PROPERTY PUBLIC p_PosR : REAL
GET
p_PosR := _Pos_R;
END_GET
END_PROPERTY

PROPERTY PUBLIC p_PosW : REAL
GET
p_PosW := _Pos_W;
END_GET
END_PROPERTY

PROPERTY PUBLIC p_PosX : REAL
GET
p_PosX := _Pos_X;
END_GET
END_PROPERTY

PROPERTY PUBLIC p_PosY : REAL
GET
p_PosY := _Pos_Y;
END_GET
END_PROPERTY

PROPERTY PUBLIC p_PosZ : REAL
GET
p_PosZ := _Pos_Z;
END_GET
END_PROPERTY

PROPERTY p_ReceiveTimeout : TIME
GET
p_ReceiveTimeout := _ReceiveTimeout;
END_GET
SET
IF p_ReceiveTimeout > T#100MS AND p_ReceiveTimeout <  T#60S THEN
	_ReceiveTimeout := p_ReceiveTimeout;
ELSE
	_ReceiveTimeout := T#1S;					// default value
END_IF
END_SET
END_PROPERTY

PROPERTY p_RemoteHost : STRING
GET
p_RemoteHost := _RemoteHost;
END_GET
SET
_RemoteHost := p_RemoteHost;
END_SET
END_PROPERTY

PROPERTY p_RemotePort : UDINT
GET
p_RemotePort := _RemotePort;
END_GET
SET
_RemotePort := p_RemotePort;
END_SET
END_PROPERTY

PROPERTY p_Results : ARRAY [1..10] OF STRING
GET
p_Results := _Results;
END_GET
SET
_Results := p_Results;
END_SET
END_PROPERTY

PROPERTY p_SavePath : STRING(255)
GET
p_SavePath := _SavePath;
END_GET
SET
_SavePath := p_SavePath;
END_SET
END_PROPERTY

PROPERTY p_SendTimeout : TIME
GET
p_SendTimeout := _SendTimeout;
END_GET
SET
IF p_SendTimeout > T#100MS AND p_SendTimeout <  T#60S THEN
	_SendTimeout := p_SendTimeout;
ELSE
	_SendTimeout := T#1S;					// default value
END_IF
END_SET
END_PROPERTY

METHOD ReadSequence : BOOL
VAR_INPUT
	sRequest		:REFERENCE TO STRING;
	sResponse		:REFERENCE TO STRING;
	nErrorId		:REFERENCE TO UDINT;
END_VAR
TCP_Com();
ReadSequence := FALSE;
CASE nReadSeqStep OF
0:		fbConnect.bExecute := TRUE;
		sResponse := '';
		nReadSeqStep := nReadSeqStep + 20;
	
20:		IF NOT fbConnect.bBusy THEN
			fbConnect.bExecute := FALSE;
			nReadSeqStep := nReadSeqStep + 20;
		ELSIF fbConnect.bError THEN
			sResponse := '';
			nErrorId := fbConnect.nErrId;
			fbConnect.bExecute := FALSE;
			nReadSeqStep := 200;
		END_IF
	
40:		sTxBuffer := sRequest;
		fbSend.bExecute := TRUE;
		nReadSeqStep := nReadSeqStep + 20;
	
60:		IF NOT fbSend.bBusy THEN
			fbSend.bExecute := FALSE;
			nReadSeqStep := 100;
		ELSIF fbSend.bError THEN
			sResponse := '';
			nErrorId := fbSend.nErrId;
			fbSend.bExecute := FALSE;
			nReadSeqStep := 200;
		END_IF
	
100:	fbReceive.bExecute := TRUE;
		nReadSeqStep := nReadSeqStep + 20;
	
120:	IF NOT fbReceive.bBusy THEN
			IF NOT fbReceive.bError THEN
					fbReceive.bExecute := FALSE;
					nReadSeqStep := nReadSeqStep + 20;
			ELSE
					sResponse := '';
					nErrorId := fbReceive.nErrId;
					fbReceive.bExecute := FALSE;
					nReadSeqStep := 200;
			END_IF
		END_IF

140:	IF fbReceive.nRecBytes > 0 THEN
			sResponse := CONCAT(sResponse, Left(sRxBuffer,UDINT_TO_INT(fbReceive.nRecBytes)));
		END_IF
		IF 		Right(sResponse, 2) = '$r$n' THEN
					nErrorId := fbReceive.nErrId;
					Delete(sResponse,2,Find(sResponse,'$r$n'));
					nReadSeqStep := 200;
		ELSIF	Right(sResponse, 1) = '$r' THEN
					nErrorId := fbReceive.nErrId;
					Delete(sResponse,1,Find(sResponse,'$r'));
					nReadSeqStep := 200;
		ELSE				
					nReadSeqStep := 100;
		END_IF
		
200:	fbClose.bExecute := TRUE;
		nReadSeqStep := nReadSeqStep + 20;
	
220:	IF NOT fbClose.bBusy THEN
			fbClose.bExecute := FALSE;
			nReadSeqStep := 500;
		ELSIF fbClose.bError THEN
			sResponse := '';
			nErrorId := fbClose.nErrId;
			fbClose.bExecute := FALSE;
			nReadSeqStep := 500;
		END_IF

500:
		ReadSequence := TRUE;
		nReadSeqStep := 0;
END_CASE
END_METHOD

METHOD ReadSR1000 : BOOL
VAR_INPUT
	sCode						:REFERENCE TO STRING;
	nErrorId					:REFERENCE TO UDINT;
END_VAR
TCP_Com();
ReadSR1000 := FALSE;

CASE nCamCheckStep OF
0:		sRequest := 'LON$R$N';
		nCamCheckStep := nCamCheckStep + 20;

20:		IF ReadSequence(sRequest, sCode, nErrorId) THEN
			nCamCheckStep := nCamCheckStep + 20;
		END_IF

40:		ReadSR1000 := TRUE;
		nCamCheckStep := 0;
END_CASE
END_METHOD

METHOD ResetCam : BOOL
VAR_INPUT
END_VAR
nCamCheckStep := 0;
END_METHOD

METHOD PRIVATE TCP_Com : BOOL
VAR_INPUT
END_VAR
fbConnect(
	sSrvNetId:= '', 
	sRemoteHost:= _RemoteHost, 
	nRemotePort:= _RemotePort, 
	bExecute:= , 
	tTimeout:= _ConnectTimeout, 
	bBusy=> , 
	bError=> , 
	nErrId=> , 
	hSocket=> );
	
fbSend(
	sSrvNetId:= '', 
	hSocket:= fbConnect.hSocket, 
	cbLen:= INT_TO_UDINT(LEN(sTxBuffer)), 
	pSrc:= ADR(sTxBuffer), 
	bExecute:= , 
	tTimeout:= _SendTimeout, 
	bBusy=> , 
	bError=> , 
	nErrId=> );

fbReceive(
	sSrvNetId:= '', 
	hSocket:= fbConnect.hSocket, 
	cbLen:= SIZEOF(sRxBuffer), 
	pDest:= ADR(sRxBuffer), 
	bExecute:= , 
	tTimeout:= _ReceiveTimeout, 
	bBusy=> , 
	bError=> , 
	nErrId=> , 
	nRecBytes=> );

fbClose(
	sSrvNetId:= '', 
	hSocket:= fbConnect.hSocket, 
	bExecute:= , 
	tTimeout:= , 
	bBusy=> , 
	bError=> , 
	nErrId=> );
END_METHOD

END_FUNCTION_BLOCK

// ---- POUs/FBs/ID200/FB_ID200.TcPOU
FUNCTION_BLOCK FB_ID200
VAR_INPUT
	
END_VAR
VAR_OUTPUT
	
END_VAR
VAR
	arrDataIn		AT %I*		: ARRAY [0..63] OF BYTE;
	arrDataOut		AT %Q*		: ARRAY [0..63] OF BYTE;
	PnIoBoxState	AT %I*		: UINT;
END_VAR
VAR
	_ch1_tag_data				: ST_Tag_Data;
	_ch2_tag_data				: ST_Tag_Data;
END_VAR
VAR
	Channel			: BYTE;
	TagData			: ST_Tag_Data;
	RawData			: RawToUlint;
END_VAR

ChkData();

PROPERTY PUBLIC Ch1_TagData : ST_Tag_Data
GET
Ch1_TagData := _ch1_tag_data;
END_GET
SET
_ch1_tag_data := Ch1_TagData;
END_SET
END_PROPERTY

PROPERTY PUBLIC Ch2_TagData : ST_Tag_Data
GET
Ch2_TagData := _ch2_tag_data;
END_GET
SET
_ch2_tag_data := Ch2_TagData;
END_SET
END_PROPERTY

METHOD PUBLIC ChangeTag : BOOL
VAR_INPUT
	Channel				: BYTE;
	CarrierType			: E_CarrierType;
END_VAR
VAR
	temp				: WordToBytes;
END_VAR
// Set command
arrDataOut[0] := E_Command.ChangeTag;

//Set Channel
arrDataOut[1].1 := Channel.0;
arrDataOut[1].2 := Channel.1;
arrDataOut[1].3 := Channel.2;
arrDataOut[1].4 := 0;
arrDataOut[1].5 := 0;
arrDataOut[1].6 := 0;
arrDataOut[1].7 := 0;

//Set Carrier type
temp.word_in := CarrierType;
arrDataOut[2] := temp.bytes[1];
arrDataOut[3] := temp.bytes[0];

//Start! Set toggle bit.
IF (arrDataIn[1].0 = arrDataOut[1].0) AND (arrDataIn[0] <> arrDataOut[0]) THEN
	MEMSET(ADR(arrDataOut)+4, 16#00, SIZEOF(arrDataOut)-4);
	arrDataOut[1].0 := NOT arrDataOut[1].0;
END_IF

ChangeTag :=		arrDataIn[0] = arrDataOut[0] AND
					arrDataIn[1] = arrDataOut[1] AND
					arrDataIn[2] = 0;
END_METHOD

METHOD PRIVATE ChkData : BOOL
VAR
//	Channel			: BYTE;
//	TagData			: ST_Tag_Data;
//	RawData			: RawToUlint;
END_VAR
Channel := 0;
Channel.0 := arrDataIn[1].1;
Channel.1 := arrDataIn[1].2;
Channel.2 := arrDataIn[1].3;
TagData.RawData[4] := arrDataIn[4];
TagData.RawData[3] := arrDataIn[5];
TagData.RawData[2] := arrDataIn[6];
TagData.RawData[1] := arrDataIn[7];
TagData.RawData[0] := arrDataIn[8];
RawData.Raw := TagData.RawData;
TagData.Code := RawData.Number;

IF (arrDataIn[0] = 16#1D) OR (arrDataIn[0] = 16#01) THEN
	IF arrDataIn[2] = 0 THEN
		TagData.Status := E_TagStatus.FixCode;
	ELSE
		TagData.Status := E_TagStatus.NotPresent;
	END_IF
	IF Channel = 1 THEN
		_ch1_tag_data := TagData;
	ELSIF Channel = 2 THEN
		_ch2_tag_data := TagData;
	END_IF
ELSIF (arrDataIn[0] = 16#10) OR (arrDataIn[0] = 16#19) THEN
	IF arrDataIn[2] = 0 THEN
		TagData.Status := E_TagStatus.UserCode;
	ELSE
		TagData.Status := E_TagStatus.NotPresent;
	END_IF
	IF Channel = 1 THEN
		_ch1_tag_data := TagData;
	ELSIF Channel = 2 THEN
		_ch2_tag_data := TagData;
	END_IF
END_IF
END_METHOD

METHOD PUBLIC EncReadFixCode : BOOL
VAR_INPUT
	Channel				:BYTE;
END_VAR
// Set command
arrDataOut[0] := E_Command.EnchancedReadFixCode;

//Set Channel
arrDataOut[1].1 := Channel.0;
arrDataOut[1].2 := Channel.1;
arrDataOut[1].3 := Channel.2;
arrDataOut[1].4 := 0;
arrDataOut[1].5 := 0;
arrDataOut[1].6 := 0;
arrDataOut[1].7 := 0;

//Start! Set toggle bit.
IF (arrDataIn[1].0 = arrDataOut[1].0) AND (arrDataIn[0] <> arrDataOut[0]) THEN
	MEMSET(ADR(arrDataOut)+2, 16#00, SIZEOF(arrDataOut)-2);
	arrDataOut[1].0 := NOT arrDataOut[1].0;
END_IF

EncReadFixCode :=		arrDataIn[0] = arrDataOut[0] AND
						arrDataIn[1] = arrDataOut[1] AND
						(arrDataIn[2] = 0 OR arrDataIn[2] = 5);
END_METHOD

METHOD PUBLIC EncReadWords : BOOL
VAR_INPUT
	Channel				:BYTE;
	WordNr				:BYTE;
END_VAR
// Set command
arrDataOut[0] := E_Command.EnchancedReadWords;

//Set Channel
arrDataOut[1].1 := Channel.0;
arrDataOut[1].2 := Channel.1;
arrDataOut[1].3 := Channel.2;

//Set WordNr
arrDataOut[1].4 := WordNr.0;
arrDataOut[1].5 := WordNr.1;
arrDataOut[1].6 := WordNr.2;
arrDataOut[1].7 := WordNr.3;


//Start! Set toggle bit.
IF (arrDataIn[1].0 = arrDataOut[1].0) AND (arrDataIn[0] <> arrDataOut[0]) THEN
	MEMSET(ADR(arrDataOut)+2, 16#00, SIZEOF(arrDataOut)-2);
	arrDataOut[1].0 := NOT arrDataOut[1].0;
END_IF

EncReadWords :=			arrDataIn[0] = arrDataOut[0] AND
						(arrDataIn[1] AND 16#0F) = (arrDataOut[1] AND 16#0F) AND
						(arrDataIn[2] = 0 OR arrDataIn[2] = 5);
END_METHOD

METHOD PUBLIC Quit : BOOL
VAR_INPUT
	Channel				:BYTE;
END_VAR
// Set command
arrDataOut[0] := E_Command.Quit;

//Set Channel
arrDataOut[1].1 := Channel.0;
arrDataOut[1].2 := Channel.1;
arrDataOut[1].3 := Channel.2;
arrDataOut[1].4 := 0;
arrDataOut[1].5 := 0;
arrDataOut[1].6 := 0;
arrDataOut[1].7 := 0;


//Start! Set toggle bit.
IF (arrDataIn[1].0 = arrDataOut[1].0) AND (arrDataIn[0] <> arrDataOut[0]) THEN
	MEMSET(ADR(arrDataOut)+2, 16#00, SIZEOF(arrDataOut)-2);
	arrDataOut[1].0 := NOT arrDataOut[1].0;
END_IF

Quit :=		arrDataIn[0] = arrDataOut[0] AND
			arrDataIn[1] = arrDataOut[1] AND
			arrDataIn[2] = 0;
END_METHOD

METHOD PUBLIC Reset : BOOL
VAR_INPUT
END_VAR
// Set command
arrDataOut[0] := E_Command.Reset;

//Start! Set toggle bit.
IF (arrDataIn[1].0 = arrDataOut[1].0) AND (arrDataIn[0] <> arrDataOut[0]) AND arrDataIn[0] <> 0 and arrDataIn[2] <> 16#FF THEN
		MEMSET(ADR(arrDataOut)+2, 16#00, SIZEOF(arrDataOut)-2);
		arrDataOut[1].0 := NOT arrDataOut[1].0;
END_IF

IF arrDataIn[2] = 16#FF THEN
	arrDataOut[0] := 0;
	arrDataOut[1] := 0;
	Reset := TRUE;
ELSE
	Reset := FALSE;
END_IF
END_METHOD

METHOD PUBLIC SinWriteFixCode : BOOL
VAR_INPUT
	Channel				: BYTE;
	Data				: ARRAY [0..4] OF BYTE;
END_VAR
VAR

END_VAR

// Set command
arrDataOut[0] := E_Command.SingleWriteFixCode;

// Set Channel
arrDataOut[1].1 := Channel.0;
arrDataOut[1].2 := Channel.1;
arrDataOut[1].3 := Channel.2;

//Set FixLen - 0101 -> 5
arrDataOut[1].4 := 1; //1
arrDataOut[1].5 := 0; //0
arrDataOut[1].6 := 1; //1
arrDataOut[1].7 := 0; //0

//Set Carrier type
arrDataOut[2] := 16#30;
arrDataOut[3] := 16#32;

// Set Data
MEMCPY(destAddr := ADR(arrDataOut), srcAddr :=ADR(Data), n := 5);

//Start! Set toggle bit.
IF (arrDataIn[1].0 = arrDataOut[1].0) AND (arrDataIn[0] <> arrDataOut[0]) THEN
	MEMSET(ADR(arrDataOut)+2, 16#00, SIZEOF(arrDataOut)-2);
	arrDataOut[1].0 := NOT arrDataOut[1].0;
END_IF

//SinWriteFixCode :=			arrDataIn[0] = arrDataOut[0] AND
//						(arrDataIn[1] AND 16#0F) = (arrDataOut[1] AND 16#0F) AND
//						(arrDataIn[2] = 0 OR arrDataIn[2] = 5);
						
SinWriteFixCode :=			arrDataIn[0] = arrDataOut[0] AND
						arrDataIn[1] = arrDataOut[1] AND
						arrDataIn[2] = 0;
END_METHOD

METHOD PUBLIC SinWriteWords : BOOL
VAR_INPUT
	Channel				:	BYTE;
	WordNr				:	BYTE;
	//WordNr				:	UINT;
	Data				: 	ARRAY [0..7] OF BYTE;
	DataLength			: 	UINT;
END_VAR
// Set command
arrDataOut[0] := E_Command.SingleWriteWords;

//Set Channel
arrDataOut[1].1 := Channel.0;
arrDataOut[1].2 := Channel.1;
arrDataOut[1].3 := Channel.2;

//Set WordNr
arrDataOut[1].4 := WordNr.0;
arrDataOut[1].5 := WordNr.1;
arrDataOut[1].6 := WordNr.2;
arrDataOut[1].7 := WordNr.3;

//Set Data

MEMCPY(destAddr := ADR(arrDataOut)+4, srcAddr :=ADR(Data), n := DataLength);

//arrDataOut[4] := Data[0];
//arrDataOut[5] := Data[1];
//arrDataOut[6] := Data[2];
//arrDataOut[7] := Data[3];


//Start! Set toggle bit.
IF (arrDataIn[1].0 = arrDataOut[1].0) AND (arrDataIn[0] <> arrDataOut[0]) THEN
	MEMSET(ADR(arrDataOut)+2, 16#00, SIZEOF(arrDataOut)-2);
	arrDataOut[1].0 := NOT arrDataOut[1].0;
END_IF

SinWriteWords :=			arrDataIn[0] = arrDataOut[0] AND
						(arrDataIn[1] AND 16#0F) = (arrDataOut[1] AND 16#0F) AND
						(arrDataIn[2] = 0 OR arrDataIn[2] = 5);
END_METHOD

END_FUNCTION_BLOCK

// ---- POUs/FBs/AWEA/FB_AWEA.TcPOU
FUNCTION_BLOCK FB_AWEA
VAR_INPUT
END_VAR
VAR_OUTPUT
END_VAR
VAR
	DigIn		AT %I*		:ST_AWEA_In;
	DigOut		AT %Q*		:ST_AWEA_Out;
END_VAR

END_FUNCTION_BLOCK

// ---- POUs/FBs/FB_Server.TcPOU
FUNCTION_BLOCK FB_Server
VAR_INPUT
END_VAR
VAR_OUTPUT
END_VAR
VAR
	fbConnect 					:FB_ServerClientConnection;
	fbSocketReceive				:FB_SocketReceive;
	fbSocketSend				:FB_SocketSend;
	hServer						:T_HSERVER;
	hSocket						:T_HSOCKET;
	buffer						:ARRAY[0..1000] OF BYTE;
	cbReceived					:UDINT;
	fbTimeoutReceive			:TON;						//Disconnect if no data was sent for an interval
	
	//HMI
	sRemoteAddress				:STRING;
	sLastConTime				:STRING(8);	
	bClientConnected			:BOOL;	
	bInit						:BOOL;					
	
	//Properties
	_SrvNetID					:STRING;
	_Host						:T_IPv4Addr;				
	_Port						:UDINT;						
	_Timeout					:TIME;
	_Timestamp					:STRING(8);
	_SystemTime					:DATE_AND_TIME;	
	_SocketState				:E_SocketConnectionState;
	_ReceivedData				:ARRAY[0..1000] OF BYTE;	
END_VAR

_SocketState := fbConnect.eState;
fbTimeoutReceive(IN:= fbTimeoutReceive.IN, PT:= _Timeout);

// HMI
bClientConnected := IsSocketAlive();
IF bInit THEN
	Init(sSrvNetID, sLocalHost, nLocalPort, nTimeoutInSeconds);
	bInit := FALSE;
END_IF

METHOD AcceptConnection : BOOL
VAR_INPUT
END_VAR
AcceptConnection := FALSE;
fbConnect(
	hServer:= hServer, 
	eMode:= eACCEPT_ALL, 
	bEnable:= TRUE, 
	tReconnect:= T#1S, 
	hSocket=> hSocket);
	
IF NOT fbConnect.bBusy AND NOT fbConnect.bError AND fbConnect.eState = eSOCKET_CONNECTED THEN
	sRemoteAddress := SOCKETADDR_TO_STRING(hSocket.remoteAddr);
	sLastConTime := _Timestamp;
	AcceptConnection := TRUE;
ELSIF fbConnect.bError THEN
	AcceptConnection := TRUE;
END_IF
END_METHOD

METHOD CloseConnection : BOOL
VAR_INPUT
END_VAR
fbConnect(
	hServer:= hServer, 
	bEnable:= FALSE);
CloseConnection := TRUE;
END_METHOD

PROPERTY Host : T_IPv4Addr
GET
Host := _Host;
END_GET
END_PROPERTY

METHOD Init : BOOL
VAR_INPUT
	sSrvNetID					:T_AmsNetID	:= '';	
	sLocalHost					:T_IPv4Addr	:= '127.0.0.0';		(* Own (server) IP address! *)
	nLocalPort					:UDINT 		:= 15000;			(* Own (server) port number! *)
	nTimeoutInSeconds			:UINT 		:= 5;
END_VAR
Init := F_CreateServerHnd(
		sSrvNetID 	:= sSrvNetID,
		sLocalHost 	:= sLocalHost,
		nLocalPort	:= nLocalPort,
		nMode 		:= LISTEN_MODE_CLOSEALL,
		bEnable 	:= FALSE,
		hServer 	:= hServer );
_Host := sLocalHost;
_Port := nLocalPort;
_SrvNetID := sSrvNetID;
_Timeout := UINT_TO_TIME(nTimeoutInSeconds * 1000);
END_METHOD

METHOD IsSocketAlive : BOOL
VAR_INPUT
END_VAR
IsSocketAlive := _SocketState = E_SocketConnectionState.eSOCKET_CONNECTED;
END_METHOD

PROPERTY Port : UDINT
GET
Port := _Port;
END_GET
END_PROPERTY

METHOD Receive : BOOL
VAR_INPUT
	pData			:POINTER TO BYTE;	// Pointer to data
	nDataSize		:UDINT;				// Size of the data
END_VAR
Receive := FALSE;
IF _SocketState = E_SocketConnectionState.eSOCKET_CONNECTED THEN
	fbSocketReceive(
	sSrvNetId:= _SrvNetID, 
	hSocket:= hSocket, 
	cbLen:= SIZEOF(buffer), 
	pDest:= ADR(buffer), 
	bExecute:= TRUE, 
	tTimeout:= _Timeout);
	
	IF NOT fbSocketReceive.bBusy THEN
		fbSocketReceive(bExecute := FALSE);
		IF fbSocketReceive.nRecBytes <> 0 THEN
			cbReceived := fbSocketReceive.nRecBytes;
			MEMSET(ADR(_ReceivedData), 0, SIZEOF(_ReceivedData));
			MEMCPY(ADR(_ReceivedData), ADR(buffer), cbReceived);
			MEMSET(pData, 0, nDataSize);
			MEMCPY(pData, ADR(buffer), cbReceived);
			MEMSET(ADR(buffer),0,cbReceived);
			fbTimeoutReceive.IN := FALSE;
			Receive := TRUE;
		ELSE
			fbTimeoutReceive.IN := TRUE;
		END_IF
	END_IF
	IF fbSocketReceive.bError THEN
		CloseConnection();
		Receive := TRUE;
	END_IF
END_IF

IF fbTimeoutReceive.Q THEN
	fbTimeoutReceive.IN := FALSE;
	fbSocketReceive(bExecute := FALSE);
	CloseConnection();
	Receive := TRUE;
END_IF
END_METHOD

METHOD Send : BOOL
VAR_INPUT
	pData			:POINTER TO BYTE;	// Pointer to data
	nDataSize		:UDINT;				// Size of the data
END_VAR
Send := FALSE;
IF _SocketState = E_SocketConnectionState.eSOCKET_CONNECTED THEN
	fbSocketSend(
			sSrvNetId:= _SrvNetID, 
			hSocket:= hSocket, 
			cbLen:= nDataSize, 
			pSrc:= pData, 
			bExecute:= TRUE, 
			tTimeout:= _Timeout);
			
	IF NOT fbSocketSend.bBusy THEN
		fbSocketSend(bExecute := FALSE);
		Send := TRUE;
	END_IF
	IF fbSocketSend.bError THEN
		CloseConnection();
		Send := TRUE;
	END_IF
END_IF
END_METHOD

PROPERTY SocketState : E_SocketConnectionState
GET
SocketState := _SocketState;
END_GET
END_PROPERTY

PROPERTY SystemTime : DATE_AND_TIME
SET
_SystemTime := SystemTime;
END_SET
END_PROPERTY

PROPERTY Timeout : TIME
GET
Timeout := _Timeout;
END_GET
END_PROPERTY

PROPERTY Timestamp : STRING
SET
_Timestamp := Timestamp;
END_SET
END_PROPERTY

END_FUNCTION_BLOCK

// ---- POUs/FBs/MySQL/SetViseState/FB_SP_spSetViseStae.TcPOU
FUNCTION_BLOCK FB_SP_spSetViseStae
VAR_INPUT
	Target						: BYTE;		// 0:empty;		1:wait operator;		4,5: wait cnc;
	nRecordStartIndex			: UDINT;
	tTimeout					: TIME;
	bExecute					: BOOL;
END_VAR
VAR_OUTPUT
	bBusy						: BOOL;
	bError						: BOOL;
	ipResult					: I_TcMessage;
	nViseNr						: BYTE;
END_VAR
VAR
	R_TRIG_Execute				: R_TRIG;
	nState						: INT;
	nErrState					: INT;
	fbSQLDatabase				: FB_SQLDatabaseEvt(sNetID := '', tTimeout := TIME#5s0ms);
	fbSQLStoredProcedure		: FB_SQLStoredProcedureEvt(sNetID := '', tTimeout := TIME#5s0ms);
	fbSQLResult					: FB_SQLResultEvt(sNetID := '', tTimeout := TIME#5s0ms);
	arrParaInfo					: ARRAY[0..1] OF ST_SQLSPParameter;
	stParameterValues			: ST_ParaVal_GetNextVise;
END_VAR

CASE nState OF
	0:
		R_TRIG_Execute(CLK:=bExecute);
		IF R_TRIG_Execute.Q THEN
			nState := 1;
			bBusy:=TRUE;
			bError:=FALSE;
			nErrState:=0;
		END_IF
	1:
		IF fbSQLDatabase.Connect(1) THEN
			ipResult:=fbSQLDatabase.ipTcResult;
			IF fbSQLDatabase.bError THEN
				nErrState:=1;
				nState:=255;
			ELSE
				arrParaInfo[0].sParameterName := 'Target';
				arrParaInfo[0].eParameterType := E_SPParameterType.Input;
				arrParaInfo[0].eParameterDataType := E_ColumnType.TinyInt;
				arrParaInfo[0].nParameterSize := 1;

				arrParaInfo[1].sParameterName := 'ViseNumber';
				arrParaInfo[1].eParameterType := E_SPParameterType.Output;
				arrParaInfo[1].eParameterDataType := E_ColumnType.TinyInt;
				arrParaInfo[1].nParameterSize := 1;
				nState:= 2;
			END_IF
		END_IF
	2:
		IF fbSQLDatabase.CreateSP('spSetViseStae', ADR(arrParaInfo), SIZEOF(arrParaInfo), ADR(fbSQLStoredProcedure)) THEN
			IF fbSQLDatabase.bError THEN
				nErrState:=2;
				nState:=255;
			ELSE
				nState:=3;
			END_IF
		END_IF
	3:
		stParameterValues.Target := Target;
		IF fbSQLStoredProcedure.ExecuteDataReturn(ADR(stParameterValues), SIZEOF(stParameterValues), ADR(fbSQLResult))THEN
			ipResult:=fbSQLStoredProcedure.ipTcResult;
			IF fbSQLStoredProcedure.bError THEN
				nErrState:=3;
				nState:=255;
			ELSE
				nState:= 4;
			END_IF
		END_IF
	4:
		IF fbSQLResult.Read(nRecordStartIndex, 1, ADR(nViseNr), SIZEOF(nViseNr), TRUE, TRUE) THEN
			ipResult:=fbSQLResult.ipTcResult;
			IF fbSQLResult.bError THEN
				nErrState:=4;
				nState:= 255;
			ELSE
				nState:= 5;
			END_IF
		END_IF
	5:
		IF fbSQLStoredProcedure.Release() THEN
			IF fbSQLStoredProcedure.bError THEN
				nErrState:=5;
				nState:=255;
			ELSE
				nState:= 200;
			END_IF
		END_IF
	200:
		IF fbSQLDatabase.Disconnect() THEN
			nState := 0;
			bBusy:= FALSE;
		END_IF
	255:
		bError:= TRUE;
		bBusy:= FALSE;
		IF nErrState > 1 THEN
			nState:=200;
		ELSE
			nState:=0;
		END_IF
END_CASE

END_FUNCTION_BLOCK

// ---- POUs/FBs/Utilities/FB_FullCycleTime.TcPOU
FUNCTION_BLOCK FB_FullCycleTime
VAR_INPUT
	bPalletSensor			:BOOL;
	timTimeMax				:TIME:= T#120S;
END_VAR
VAR_OUTPUT
	nCurrentCycleTime		:REAL;
	arrCycleTimes			:ARRAY [1..10] OF REAL;
END_VAR
VAR
	tCycleTime				:TON;
	rStart					:R_TRIG;
END_VAR

rStart(CLK:= bPalletSensor);
tCycleTime(IN:= TRUE, PT:= timTimeMax);

IF 		rStart.Q THEN
				MEMMOVE(ADR(arrCycleTimes)+4,ADR(arrCycleTimes),SIZEOF(arrCycleTimes)-4);
				arrCycleTimes[1] := nCurrentCycleTime;
				tCycleTime(IN:= FALSE);
ELSIF	NOT tCycleTime.Q THEN
				nCurrentCycleTime := (TIME_TO_REAL(tCycleTime.ET) / 1000);
ELSE
				nCurrentCycleTime := (TIME_TO_REAL(timTimeMax) / 1000);
END_IF

END_FUNCTION_BLOCK

// ---- POUs/FBs/Utilities/FB_TcEvent.TcPOU
FUNCTION_BLOCK FB_TcEvent
VAR_INPUT
	sName							:STRING;
	stPosData						:ST_PosData;
	bAck							:BOOL;
	stEventEntry					:TcEventEntry;				(*Event definition*)
	aErrorDesc					:ARRAY [0..31] OF STRING;
END_VAR
VAR_OUTPUT
	sError						:STRING(255);					(*hiba string*)
END_VAR
VAR
	i							:INT;
	nErrorCodeTmp				:UDINT;
	bIsInitalized				:BOOL;
	fbAlarm						:FB_TcAlarm;
	fbErrorRTrig				:R_Trig;
	fbAckRTrig					:R_Trig;
END_VAR

IF stPosData.bError THEN
	sError := sName;
	nErrorCodeTmp :=  stPosData.nErrorCode;
	FOR i:=0 TO 31 DO
		IF nErrorCodeTmp.0 THEN
			sError :=  CONCAT(sError, aErrorDesc[i]);
		END_IF
		nErrorCodeTmp := SHR(nErrorCodeTmp,1);
	END_FOR
ELSE
	sError := '';
END_IF

(*Hiba kezelés Tc3_EventLogger*)
IF NOT bIsInitalized THEN
	bIsInitalized := TRUE;
	fbAlarm.CreateEx(stEventEntry, TRUE, 0);
END_IF

fbErrorRTrig(CLK:= stPosData.bError);
fbAckRTrig(CLK:= bAck);

(*Hiba generálás*)
IF fbErrorRTrig.Q THEN
	fbAlarm.ipArguments.Clear().AddString(sError);
	fbAlarm.Raise(0);
END_IF
(*Hiba nyugtázás*)
IF fbAckRTrig.Q THEN
	fbAlarm.Confirm(0);
END_IF
(*Hiba törlés (nyugtázott és megszűnt)*)
IF fbAlarm.eConfirmationState = 3 AND NOT stPosData.bError THEN
	fbAlarm.Clear(0, FALSE);
END_IF

END_FUNCTION_BLOCK

// ---- POUs/FBs/Utilities/FB_UpsC69xx.TcPOU
FUNCTION_BLOCK FB_UpsC69xx
VAR_INPUT
	bEnable					:BOOL;					// FB Engedély.
	tShdnTime				:TIME := T#10S;			// Tápkimaradási időkorlát
	nShdnDelay				:DWORD := 0;			// Leállítási késleltetés
END_VAR
VAR_OUTPUT
	bPowerOK				:BOOL;					// Tápellátás rendben
	nBatteryLife			:DWORD;					// Akkumulátor állapot (százalékba)
	bError					:BOOL;					// Hiba bit
	nErrId					:UDINT;					// Hiba kód
END_VAR
VAR
	fbGetUpsStatus			:FB_GetUPSStatus;
	ntShutdown				:NT_Shutdown;
	tShutdown				:TON;
END_VAR

(*-----=== UPS ===-----*)
(*	--------------------------------------------------------------------------------
	Leírás		:	C69XX CPU Szünetmentes táp kezelés
	Név			:	FB_UpsC69xx
	Módosító	:	Závori Zsolt
	Dátum		:	2019.07.05
	Revízió		:	1.0
	--------------------------------------------------------------------------------
	Feltételek	:	Tc2_Utilities-(REF), Tc2_IoFunctions
	Változók	:	-
	Visu		:	-
	UserControl	:	-
	--------------------------------------------------------------------------------
	Részletek	:	-					
*)
fbGetUpsStatus(bEnable:= bEnable );
fbGetUpsStatus( 
	bEnable:= bEnable, 
	bError=> bError, 
	nErrId=> nErrId);

nBatteryLife := fbGetUpsStatus.stStatus.BatteryLifePercent;

tShutdown(
		IN:= fbGetUpsStatus.stStatus.ePowerStatus = PowerOnBattery AND
			 fbGetUpsStatus.bValid AND NOT fbGetUpsStatus.bError AND bEnable,
		PT:= tShdnTime);

bPowerOK := (fbGetUpsStatus.stStatus.ePowerStatus = PowerOnLine);		
IF tShutdown.Q THEN
	ntShutdown(
			DELAY:= nShdnDelay, 
			START:= TRUE);
END_IF

END_FUNCTION_BLOCK

// ---- POUs/FBs/Utilities/FB_UserLed.TcPOU
FUNCTION_BLOCK FB_UserLed
VAR_INPUT
	bEnable					:BOOL;					// FB Engedély.
	eULedColor				:E_UsrLED_Color;
END_VAR
VAR_OUTPUT
	bError					:BOOL;					// Hiba bit
	nErrId					:UDINT;					// Hiba kód
END_VAR
VAR
	fbUserLED				:FB_SetLedColor_BAPI;
END_VAR

(*-----=== User LED ===-----*)
(*	--------------------------------------------------------------------------------
	Leírás		:	C69XX CPU User LED kezelés
	Név			:	FB_UserLed
	Módosító	:	Závori Zsolt
	Dátum		:	2019.07.05
	Revízió		:	1.0
	--------------------------------------------------------------------------------
	Feltételek	:	Tc2_IoFunctions
	Változók	:	-
	Visu		:	-
	UserControl	:	-
	--------------------------------------------------------------------------------
	Részletek	:	-					
*)
IF		fbUserLED.eNewColor <> eULedColor AND
		NOT fbUserLED.bExecute AND
		NOT fbUserLED.bBusy THEN
			fbUserLED.eNewColor := eULedColor;
			fbUserLED.bExecute := TRUE;
ELSIF	(fbUserLED.bExecute AND NOT fbUserLED.bBusy) OR fbUserLED.bError THEN
			fbUserLED.bExecute := FALSE;
END_IF
fbUserLED();
bError := fbUserLED.bError;
nErrId := fbUserLED.nErrID;

END_FUNCTION_BLOCK

// ---- POUs/FBs/Utilities/FB_WorkLight.TcPOU
FUNCTION_BLOCK FB_WorkLight
VAR_INPUT
	bDoorClose					:BOOL;
	bManualCtrl					:BOOL;
	nEcoTime					:UINT := 5;
END_VAR
VAR_OUTPUT
	bLightCtrl					:BOOL;
END_VAR
VAR
	tEcoTime					:TON;
	rtDoorOn					:R_Trig;
	rtManualOn					:R_Trig;
	rtDoorOff					:R_Trig;
	rtManualOff					:R_Trig;
	rtTimerOff					:R_Trig;
END_VAR

rtDoorOn(CLK:= NOT bDoorClose);
rtManualOn(CLK:= bManualCtrl);
rtDoorOff(CLK:= bDoorClose);
rtManualOff(CLK:= NOT bManualCtrl);
rtTimerOff(CLK:= tEcoTime.Q);
tEcoTime(IN:= bLightCtrl, PT:= (nEcoTime * T#1M));

IF rtDoorOn.Q OR rtManualOn.Q THEN
	bLightCtrl := TRUE;
	bManualCtrl := TRUE;
END_IF

IF rtDoorOff.Q OR rtManualOff.Q OR rtTimerOff.Q THEN
	bLightCtrl := FALSE;
	bManualCtrl := FALSE;
END_IF

END_FUNCTION_BLOCK

// ---- POUs/InitTCPIP.TcPOU
PROGRAM InitTCPIP
VAR
	sSrvNetID 		: T_AmsNetID := '';(* TwinCAT TCP/IP server network address *)
	fbCloseAll		: FB_SocketCloseAll;
END_VAR

(* On PLC reset or program download close all created/opened sockets/connections *)
fbCloseAll( sSrvNetID := sSrvNetID, bExecute:= bInitTCPIP );
IF fbCloseAll.bBusy OR fbCloseAll.bError THEN
	RETURN;
END_IF
bInitTCPIP := FALSE;

END_PROGRAM

// ---- POUs/Temp/FB_ContiRobot.TcPOU
FUNCTION_BLOCK FB_ContiRobot
VAR_INPUT
	nPcbType					:WORD;
	
	bPcbStat_N					:BOOL;
	bPcbStat_Pass				:BOOL;
	bPcbStat_Fail				:BOOL;
	bPcbInFixture				:BOOL;
	bPcbSensor11				:BOOL;
	bPcbSensor12				:BOOL;
	bPcbSensor21				:BOOL;
	bPcbSensor22				:BOOL;
	
	bEmy_OK						:BOOL;
	bDoor_OK					:BOOL;
	bOpDoorUp					:BOOL;
	bOpDoorDown					:BOOL;
	bDoorsClose					:BOOL;
	bDoorsLock					:BOOL;
	bEmyBtn_1					:BOOL;
	bEmyBtn_2					:BOOL;
	
	bReady						:BOOL;
	bWaitDutIn					:BOOL;
	bWaitDutOut					:BOOL;
	bError						:BOOL;
	bEcoMode					:BOOL;
	bInProcess					:BOOL;
	
	stFanucIn					:ST_Fanuc_In;
	
	nErrorCode					:WORD;
	
	bMoveAreaEnable				:BOOL;
	bDoorOpenEnable				:BOOL;

	nLifeSignalOut				:UINT;
END_VAR
VAR_OUTPUT
	bMoveAreaReq				:BOOL;
	bDoorOpenReq				:BOOL;
	bStart						:BOOL;
	
	nLifeSignalIn				:UINT;
	
END_VAR
VAR
	uConvWord					:U_WordToArrOfByte;
	Inputs_0		AT %I*		:ARRAY [0..3] OF BYTE;
	Inputs_1		AT %I*		:ARRAY [0..3] OF BYTE;
	Inputs_2		AT %I*		:ARRAY [0..3] OF BYTE;
	Inputs_3		AT %I*		:ARRAY [0..3] OF BYTE;
	Inputs_4		AT %I*		:ARRAY [0..3] OF BYTE;
	Inputs_5		AT %I*		:ARRAY [0..3] OF BYTE;
	Inputs_6		AT %I*		:ARRAY [0..3] OF BYTE;
	Inputs_7		AT %I*		:ARRAY [0..3] OF BYTE;
	

	Outputs_0		AT %Q*		:ARRAY [0..3] OF BYTE;
	Outputs_1		AT %Q*		:ARRAY [0..3] OF BYTE;
	Outputs_2		AT %Q*		:ARRAY [0..3] OF BYTE;
	Outputs_3		AT %Q*		:ARRAY [0..3] OF BYTE;
	Outputs_4		AT %Q*		:ARRAY [0..3] OF BYTE;
	Outputs_5		AT %Q*		:ARRAY [0..3] OF BYTE;
	Outputs_6		AT %Q*		:ARRAY [0..3] OF BYTE;
	Outputs_7		AT %Q*		:ARRAY [0..3] OF BYTE;
END_VAR

(* -----=== DUT type ===----- *)
Outputs_0[3] := WORD_TO_BYTE(nPcbType);				//	00.0 .. 00.7	PCBA Típusa

(* -----=== DUT status ===----- *)
Outputs_0[2].0 := bPcbStat_N;						//	01.0			PCBA állapot nem ismert
Outputs_0[2].1 := bPcbStat_Pass;					//	01.1			PCBA állapot 'Pass'
Outputs_0[2].2 := bPcbStat_Fail;					//	01.2			PCBA állapot 'Fail'
Outputs_0[2].3 := bPcbInFixture;					//	01.3			PCBA az ülékben (kiértékelt bit)
Outputs_0[2].4 := bPcbSensor11;						//	01.4			PCBA szenzor kimenet 11
Outputs_0[2].5 := bPcbSensor12;						//	01.5			PCBA szenzor kimenet 12
Outputs_0[2].6 := bPcbSensor21;						//	01.6			PCBA szenzor kimenet 21
Outputs_0[2].7 := bPcbSensor22;						//	01.7			PCBA szenzor kimenet 22

(* -----=== Safety status ===----- *)
Outputs_0[1].0 := bEmy_OK;							//	02.0			Vészkör Ok
Outputs_0[1].1 := bDoor_OK;							//	02.1			Ajtókör Ok
Outputs_0[1].2 := bOpDoorUp;						//	02.2			Operátor ajtó fent
Outputs_0[1].3 := bOpDoorDown;						//	02.3			Operátor ajtó lent
Outputs_0[1].4 := bDoorsClose;						//	02.4			Ajtók csukva
Outputs_0[1].5 := bDoorsLock;						//	02.5			Ajtók reteszelve
Outputs_0[1].6 := bEmyBtn_1;						//	02.6			Vészgomb 1
Outputs_0[1].7 := bEmyBtn_2;						//	02.7			Vészgomb 2

(* -----=== Machine status ===----- *)
Outputs_0[0].0 := bReady;							//	03.0			Az állomás üzemkész
Outputs_0[0].1 := bWaitDutIn;						//	03.1			Az állomás termék behelyezésre vár
Outputs_0[0].2 := bWaitDutOut;						//	03.2			Az állomás termék kivételre
Outputs_0[0].3 := bError;							//	03.3			Az állomás hiba állapotban van
Outputs_0[0].4 := bEcoMode;							//	03.4			Az állomás Eco állapotban van
Outputs_0[0].5 := bInProcess;						//	03.5			Az állomás folyamat közben van
//Outputs_0[0].6 := ;								//	03.6
//Outputs_0[0].7 := ;								//	03.7

(* -----=== Error code ===----- *)
uConvWord.wData := nErrorCode;
Outputs_1[3] := uConvWord.arrData[0];				//	04.0 .. 05.0	Állomás hiba kód
Outputs_1[2] := uConvWord.arrData[1];;

(* -----=== Handshake ===----- *)
Outputs_1[1].0 := bMoveAreaEnable;					//	06.0			Terület bemozgási engedély
Outputs_1[1].1 := bDoorOpenEnable;					//	06.1			Ajtónyitás engedély

//Outputs_1[0].0 := ;								//	07.01			Tartalék

(* -----=== Fanuc ===----- *)
Outputs_2[3].0 := stFanucIn.stArea.bFeeder;			//	08.0			Fanuc Area
Outputs_2[3].1 := stFanucIn.stArea.bFixtureArea;	//	08.1			Fanuc Area
Outputs_2[3].2 := stFanucIn.stArea.bPositioner1;	//	08.2			Fanuc Area
Outputs_2[3].3 := stFanucIn.stArea.bPositioner2;	//	08.3			Fanuc Area
Outputs_2[3].4 := stFanucIn.stCtrl.bBattery;		//	08.4			Fanuc Ctrl
Outputs_2[3].5 := stFanucIn.stCtrl.bBusy;			//	08.5			Fanuc Ctrl
Outputs_2[3].6 := stFanucIn.stCtrl.bCmdEnable;		//	08.6			Fanuc Ctrl
Outputs_2[3].7 := stFanucIn.stCtrl.bError;			//	08.7			Fanuc Ctrl

Outputs_2[2].0 := stFanucIn.stCtrl.bFault;			//	09.0			Fanuc Ctrl
Outputs_2[2].1 := stFanucIn.stCtrl.bProgEnd;		//	09.1			Fanuc Ctrl
Outputs_2[2].2 := stFanucIn.stCtrl.bProgRun;		//	09.2			Fanuc Ctrl
Outputs_2[2].3 := stFanucIn.stCtrl.bServiceRun;		//	09.3			Fanuc Ctrl
Outputs_2[2].4 := stFanucIn.stAlarm.bAlarm1;		//	09.4			Fanuc Alarm
Outputs_2[2].5 := stFanucIn.stAlarm.bAlarm2;		//	09.5			Fanuc Alarm
Outputs_2[2].6 := stFanucIn.stAlarm.bAlarm3;		//	09.6			Fanuc Alarm
Outputs_2[2].7 := stFanucIn.stAlarm.bAlarm4;		//	09.7			Fanuc Alarm

Outputs_2[1].0 := stFanucIn.stAlarm.bAlarm5;		//	10.0			Fanuc Alarm
Outputs_2[1].1 := stFanucIn.stAlarm.bAlarm6;		//	10.1			Fanuc Alarm
Outputs_2[1].2 := stFanucIn.stEmergency.bBEKHLD;	//	10.2			Fanuc Emergency
Outputs_2[1].3 := stFanucIn.stEmergency.bBELTBREAK;	//	10.3			Fanuc Emergency
Outputs_2[1].4 := stFanucIn.stEmergency.bEMGEX;		//	10.4			Fanuc Emergency
Outputs_2[1].5 := stFanucIn.stEmergency.bEMGOP;		//	10.5			Fanuc Emergency
Outputs_2[1].6 := stFanucIn.stEmergency.bEMGTP;		//	10.6			Fanuc Emergency
Outputs_2[1].7 := stFanucIn.stEmergency.bFALM;		//	10.7			Fanuc Emergency

Outputs_2[0].0 := stFanucIn.stEmergency.bFENCE;		//	11.0			Fanuc Emergency
Outputs_2[0].1 := stFanucIn.stEmergency.bHBK;		//	11.1			Fanuc Emergency
Outputs_2[0].2 := stFanucIn.stEmergency.bIMSTP;		//	11.2			Fanuc Emergency
Outputs_2[0].3 := stFanucIn.stEmergency.bNTED;		//	11.3			Fanuc Emergency
Outputs_2[0].4 := stFanucIn.stEmergency.bPPABN;		//	11.4			Fanuc Emergency
Outputs_2[0].5 := stFanucIn.stEmergency.bROT;		//	11.5			Fanuc Emergency
Outputs_2[0].6 := stFanucIn.stEmergency.bSRVDSCNCT;	//	11.6			Fanuc Emergency
Outputs_2[0].7 := stFanucIn.stEmergency.bSVOFF;		//	11.7			Fanuc Emergency

Outputs_3[3].0 := stFanucIn.stEmergency.bUSRALM;	//	12.0			Fanuc Emergency


(* -----=== Life signal ===----- *)
Outputs_7[0] := UINT_TO_BYTE(nLifeSignalOut);		//	63.0 .. 63.7	Életjel
{endregion}
	 
{region "Profinet -> Beckhoff"}
(* -----=== Handshake ===----- *)
bMoveAreaReq := Inputs_0[3].0;						//	00.0			Bemozgási engedély kérés
bDoorOpenReq := Inputs_0[3].1;						//	00.1			Ajtónyitás engedély kérés
bStart := Inputs_0[3].2;							//	00.1

(* -----=== Life signal ===----- *)
nLifeSignalIn := BYTE_TO_WORD(Inputs_7[0]);			//	63.0 .. 63.7	Életjel
{enregion}

END_FUNCTION_BLOCK
